TYPE E_HomeY :
(
	Init,
    Gear_In,
    Power_On,
    Check_Homed,
    Home_Y1,
    Y1_Homed,
    Home_Y2,
    Y2_Homed,
    Re_Gear,
    End_Sequence
    
);
END_TYPE

(* stored: Version 1.1.0.1, ProductVersion 3.1.4024.9
   DUT E_HomeY: Id {7737f691-b37c-43b8-aec3-3723fe7e4366} *)
